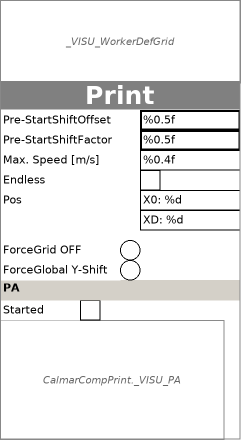
VISUALIZATION _VISU_WorkerPrint_WEU  // 241x440
VAR_IN_OUT
  m_Inst : FB_WorkerDefGrid_Print_WEU;
END_VAR
    Frame (0,0 241x83)
        shows _VISU_WorkerDefGrid(m_Inst := m_Inst)
    Rectangle (0,80 240x30), "Print", colour toggle: m_Inst._pAttachedCt <> 0
    Frame (0,320 224x120)
        shows CalmarCompPrint._VISU_PA(m_Inst := m_Inst.fbPa)
    Rectangle (0,150 120x20), "Max. Speed [m/s]"
    Rectangle (140,150 100x20), "%0.4f", text variable: m_Inst.fMaxSpeed
    Rectangle (0,170 120x20), "Endless"
    RoundedRectangle (140,170 20x20), colour toggle: m_Inst._bEndless
    Rectangle (0,300 80x20), "Started"
    RoundedRectangle (80,300 20x20), colour toggle: m_Inst._bPaStarted
    Rectangle (0,190 120x20), "Pos"
    Rectangle (140,190 100x20), "X0: %d", text variable: m_Inst._nPosX0
    Rectangle (140,210 100x20), "XD: %d", text variable: m_Inst._nPosXDelta
    Rectangle (0,280 240x20), "PA"
    Rectangle (0,240 120x20), "ForceGrid OFF"
    Ellipse (120,240 20x20), tooltip "Force Grid OFF (gridPs=0)"
        toggle m_Inst._bForceDefGridOff
    Rectangle (0,110 160x20), "Pre-StartShiftOffset"
    Rectangle (140,110 100x20), "%0.5f", text variable: m_Inst._fStartShiftOffset
        OnMouseDown: write the text variable via Default
    Rectangle (0,130 160x20), "Pre-StartShiftFactor"
    Rectangle (140,130 100x20), "%0.5f", text variable: m_Inst._fStartShiftFactor
        OnMouseDown: write the text variable via Default
    Rectangle (0,260 120x20), "ForceGlobal Y-Shift"
    Ellipse (120,260 20x20), tooltip "Force Grid OFF (gridPs=0)"
        toggle m_Inst._bForceGlobalYShift
END_VISUALIZATION

(* stored: Version 1.1.0.1, ProductVersion 3.1.4024.11
   Visu _VISU_WorkerPrint_WEU: Id {a8b82c86-7448-4902-995b-e457b2409e24} *)
